PROGRAM Automatic
VAR
	foo : BOOL;
	motor_1 : Motor;
	auto_move : AutoMove;
	auto_move_2 : AutoMove2;
	tracking : TrackingLogic;
	init : Init;
END_VAR


init();
auto_move_2();
motor_1();
tracking();

END_PROGRAM

(* stored: Version 1.1.0.1, ProductVersion 3.1.4024.12
   POU Automatic: Id {6c83d90f-8360-42e8-acf9-21e66d771135}, SpecialFunc None *)
